// TIA Portal V17 export
// export: Created 2026-04-13T11:12:42.5273063Z, ExportSetting WithDefaults, DisplayName Totally Integrated Automation Portal, DisplayVersion V17 Update 4, DisplayName TIA Portal Openness, DisplayVersion V17 Update 4, DisplayName TIA Portal Version Control Interface, DisplayVersion V17, DisplayName SINAMICS Startdrive Advanced, DisplayVersion V17, DisplayName SINAMICS Startdrive G130, G150, S120, S150, SINAMICS MV, S210, DisplayVersion V17, DisplayName SINAMICS Startdrive G110M, G120, G120C, G120D, G120P, G115D, DisplayVersion V17, DisplayName STEP 7 Professional, DisplayVersion V17 Update 4, DisplayName STEP 7 Safety, DisplayVersion V17, DisplayName WinCC Professional, DisplayVersion V17 Update 4
FUNCTION_BLOCK "0-模拟量滤波简"   // FB86, SCL
{ S7_Optimized_Access := 'TRUE' }
VERSION : 0.1
// stored: AutoNumber true, IsIECCheckEnabled false, IsRetainMemResEnabled false, MemoryReserve 100, SetENOAutomatically false, UDAEnableTagReadback false
   VAR_INPUT
      输入 : Real;   // 转换后的模拟量输入端
      采集时间 : Time := T#200ms;   // 多长时间采集一次数据，单位ms
      模式 : Bool;   // false为算数平均滤波，true为切头尾平均滤波
   END_VAR
   VAR_OUTPUT
      输出 : Real;   // 滤波后的输出值
   END_VAR
   VAR_IN_OUT
      滤波强度 : Int := 3;   // 多少个数据平均一次
   END_VAR
   VAR
      T0 : TON_TIME;
      T1 { S7_SetPoint := 'True'} : TON_TIME;
      P { S7_SetPoint := 'True'} : R_TRIG;
      最小值 { S7_SetPoint := 'True'} : Real;
      最大值 : Real;
      中间寄存数值 : Array[0..30] of Real;
   END_VAR
   VAR_TEMP
      "a" : DInt;
      "b" : DInt;
      总和 : Real;
   END_VAR
BEGIN
   REGION 初始化
       #最大值 := #中间寄存数值[1];
       #最小值 := #中间寄存数值[1];
   END_REGION


   REGION 滤波强度限制
       IF #滤波强度 < 3 THEN
           #滤波强度 := 3;
       END_IF;
       IF #滤波强度 > 30 THEN
           #滤波强度 := 30;
       END_IF;
   END_REGION


   REGION 构速时钟脉冲
       #T0(IN := NOT #T1.Q,
           PT := #采集时间 - T#20MS);
       #T1(IN :=  #T0.Q,
           PT := T#20MS);
       #P(CLK := #T0.Q);
   END_REGION

   REGION 数据写入
       IF #P.Q THEN
           FOR #a := #滤波强度 TO 2 BY -1 DO //依次将输入数据存入到寄存数组中
               #中间寄存数值[#a] := #中间寄存数值[#a - 1];
           END_FOR;
           #中间寄存数值[1] := #输入;
       END_IF;
   END_REGION


   REGION 找最值以及计算总和
       FOR #b := 1 TO #滤波强度 DO
           IF #中间寄存数值[#b] > #最大值 THEN
               #最大值 := #中间寄存数值[#b];
           END_IF;
           IF #中间寄存数值[#b] < #最小值 THEN
               #最小值 := #中间寄存数值[#b];
           END_IF;
           #总和 := #总和 + #中间寄存数值[#b]; //计算总和
       END_FOR;
   END_REGION


   REGION 求平均以及输出
       IF #模式 = TRUE THEN
           #输出 := (#总和 - #最大值 - #最小值) / DINT_TO_REAL((#滤波强度) - 2);//切尾平均滤波后输出
       ELSE
           #输出 := #总和 / DINT_TO_REAL(#滤波强度);//算数平均输出
       END_IF;
   END_REGION
END_FUNCTION_BLOCK
